// TIA Portal V20 export
DATA_BLOCK "InstStackMainDB"   // DB454
// stored: InstanceOfName 2200_StackMain, InstanceOfType FB
"2200_StackMain"
   // VAR_INPUT
   //    Calculate : Bool;
   //    SemiStep : Bool;
   //    FullStep : Bool;
   //    Auto : Bool;
   //    CycleStop : Bool;
   //    FastStop : Bool;
   //    Reset : Bool;
   //    Parameter : Struct
   //       Global : Struct
   //          CPM : LReal;
   //          StageWidth : LReal;
   //       END_STRUCT;
   //       "Step" : Struct
   //          MandrelUse : Bool;
   //          InitialPosFinalRoller : LReal;
   //          InitialPosCompensator : LReal;
   //       END_STRUCT;
   //       Auto : Struct
   //          SepaClean : Bool;
   //          CellCount : DInt;
   //          Compensator : Struct
   //             InitialPosCompensator : LReal;
   //          END_STRUCT;
   //          Anode : Struct
   //             PnPX1 : Struct
   //                InitialPosAnodePnPX1 : LReal;
   //                AnodePnPX1FwdOutputCam : Struct
   //                   OnPos : LReal;
   //                   OffPos : LReal;
   //                END_STRUCT;
   //                AnodePnPX1BwdOutputCam : Struct
   //                   OnPos : LReal;
   //                   OffPos : LReal;
   //                END_STRUCT;
   //                AnodeReelCutDataDeleteOffOutputCam : Struct
   //                   OnPos : LReal;
   //                   OffPos : LReal;
   //                END_STRUCT;
   //             END_STRUCT;
   //             PnPX2 : Struct
   //                InitialPosAnodePnPX2 : LReal;
   //                AnodePnPX2FwdOutputCam : Struct
   //                   OnPos : LReal;
   //                   OffPos : LReal;
   //                END_STRUCT;
   //                AnodePnPX2BwdOutputCam : Struct
   //                   OnPos : LReal;
   //                   OffPos : LReal;
   //                END_STRUCT;
   //             END_STRUCT;
   //             PnPZ1 : Struct
   //                InitialPosAnodePnPZ1 : LReal;
   //                AnodePnPZ1Down1OutputCam : Struct
   //                   OnPos : LReal;
   //                   OffPos : LReal;
   //                END_STRUCT;
   //                AnodePnPZ1Up1OutputCam : Struct
   //                   OnPos : LReal;
   //                   OffPos : LReal;
   //                END_STRUCT;
   //                AnodePnPZ1Down2OutputCam : Struct
   //                   OnPos : LReal;
   //                   OffPos : LReal;
   //                END_STRUCT;
   //                AnodePnPZ1Up2OutputCam : Struct
   //                   OnPos : LReal;
   //                   OffPos : LReal;
   //                END_STRUCT;
   //                AnodePnPZ1SuctionOnOutputCam : Struct
   //                   OnPos : LReal;
   //                   OffPos : LReal;
   //                END_STRUCT;
   //                AnodePnPZ1SuctionOffOutputCam : Struct
   //                   OnPos : LReal;
   //                   OffPos : LReal;
   //                END_STRUCT;
   //                AnodePnPZ1ReelCutBlowOutputCam : Struct
   //                   OnPos : LReal;
   //                   OffPos : LReal;
   //                END_STRUCT;
   //                AnodeAlignSuctionOnOutputCam : Struct
   //                   OnPos : LReal;
   //                   OffPos : LReal;
   //                END_STRUCT;
   //                AnodeReelCutDataDeleteOnOutputCam : Struct
   //                   OnPos : LReal;
   //                   OffPos : LReal;
   //                END_STRUCT;
   //                AnodeAlignVisionOutputCam : Struct
   //                   OnPos : LReal;
   //                   OffPos : LReal;
   //                END_STRUCT;
   //             END_STRUCT;
   //             PnPZ2 : Struct
   //                InitialPosAnodePnPZ2 : LReal;
   //                AnodePnPZ2Down1OutputCam : Struct
   //                   OnPos : LReal;
   //                   OffPos : LReal;
   //                END_STRUCT;
   //                AnodePnPZ2Up1OutputCam : Struct
   //                   OnPos : LReal;
   //                   OffPos : LReal;
   //                END_STRUCT;
   //                AnodePnPZ2Down2OutputCam : Struct
   //                   OnPos : LReal;
   //                   OffPos : LReal;
   //                END_STRUCT;
   //                AnodePnPZ2Up2OutputCam : Struct
   //                   OnPos : LReal;
   //                   OffPos : LReal;
   //                END_STRUCT;
   //                AnodePnPZ2SuctionOnOutputCam : Struct
   //                   OnPos : LReal;
   //                   OffPos : LReal;
   //                END_STRUCT;
   //                AnodePnPZ2SuctionOffOutputCam : Struct
   //                   OnPos : LReal;
   //                   OffPos : LReal;
   //                END_STRUCT;
   //                AnodeAlignSuctionOffOutputCam : Struct
   //                   OnPos : LReal;
   //                   OffPos : LReal;
   //                END_STRUCT;
   //             END_STRUCT;
   //          END_STRUCT;
   //          Cathode : Struct
   //             PnPX1 : Struct
   //                InitialPosCathodePnPX1 : LReal;
   //                CathodePnPX1FwdOutputCam : Struct
   //                   OnPos : LReal;
   //                   OffPos : LReal;
   //                END_STRUCT;
   //                CathodePnPX1BwdOutputCam : Struct
   //                   OnPos : LReal;
   //                   OffPos : LReal;
   //                END_STRUCT;
   //                CathodeReelCutDataDeleteOffOutputCam : Struct
   //                   OnPos : LReal;
   //                   OffPos : LReal;
   //                END_STRUCT;
   //             END_STRUCT;
   //             PnPX2 : Struct
   //                InitialPosCathodePnPX2 : LReal;
   //                CathodePnPX2FwdOutputCam : Struct
   //                   OnPos : LReal;
   //                   OffPos : LReal;
   //                END_STRUCT;
   //                CathodePnPX2BwdOutputCam : Struct
   //                   OnPos : LReal;
   //                   OffPos : LReal;
   //                END_STRUCT;
   //             END_STRUCT;
   //             PnPZ1 : Struct
   //                InitialPosCathodePnPZ1 : LReal;
   //                CathodePnPZ1Down1OutputCam : Struct
   //                   OnPos : LReal;
   //                   OffPos : LReal;
   //                END_STRUCT;
   //                CathodePnPZ1Up1OutputCam : Struct
   //                   OnPos : LReal;
   //                   OffPos : LReal;
   //                END_STRUCT;
   //                CathodePnPZ1Down2OutputCam : Struct
   //                   OnPos : LReal;
   //                   OffPos : LReal;
   //                END_STRUCT;
   //                CathodePnPZ1Up2OutputCam : Struct
   //                   OnPos : LReal;
   //                   OffPos : LReal;
   //                END_STRUCT;
   //                CathodePnPZ1SuctionOnOutputCam : Struct
   //                   OnPos : LReal;
   //                   OffPos : LReal;
   //                END_STRUCT;
   //                CathodePnPZ1SuctionOffOutputCam : Struct
   //                   OnPos : LReal;
   //                   OffPos : LReal;
   //                END_STRUCT;
   //                CathodePnPZ1ReelCutBlowOutputCam : Struct
   //                   OnPos : LReal;
   //                   OffPos : LReal;
   //                END_STRUCT;
   //                CathodeAlignSuctionOnOutputCam : Struct
   //                   OnPos : LReal;
   //                   OffPos : LReal;
   //                END_STRUCT;
   //                CathodeReelCutDataDeleteOnOutputCam : Struct
   //                   OnPos : LReal;
   //                   OffPos : LReal;
   //                END_STRUCT;
   //                CathodeAlignVisionOutputCam : Struct
   //                   OnPos : LReal;
   //                   OffPos : LReal;
   //                END_STRUCT;
   //             END_STRUCT;
   //             PnPZ2 : Struct
   //                InitialPosCathodePnPZ2 : LReal;
   //                CathodePnPZ2Down1OutputCam : Struct
   //                   OnPos : LReal;
   //                   OffPos : LReal;
   //                END_STRUCT;
   //                CathodePnPZ2Up1OutputCam : Struct
   //                   OnPos : LReal;
   //                   OffPos : LReal;
   //                END_STRUCT;
   //                CathodePnPZ2Down2OutputCam : Struct
   //                   OnPos : LReal;
   //                   OffPos : LReal;
   //                END_STRUCT;
   //                CathodePnPZ2Up2OutputCam : Struct
   //                   OnPos : LReal;
   //                   OffPos : LReal;
   //                END_STRUCT;
   //                CathodePnPZ2SuctionOnOutputCam : Struct
   //                   OnPos : LReal;
   //                   OffPos : LReal;
   //                END_STRUCT;
   //                CathodePnPZ2SuctionOffOutputCam : Struct
   //                   OnPos : LReal;
   //                   OffPos : LReal;
   //                END_STRUCT;
   //                CathodeAlignSuctionOffOutputCam : Struct
   //                   OnPos : LReal;
   //                   OffPos : LReal;
   //                END_STRUCT;
   //             END_STRUCT;
   //          END_STRUCT;
   //          FinalRoller : Struct
   //             InitialPosFinalRoller : LReal;
   //             FinalRollerFwdOutputCam : Struct
   //                OnPos : LReal;
   //                OffPos : LReal;
   //             END_STRUCT;
   //             FinalRollerBwdOutputCam : Struct
   //                OnPos : LReal;
   //                OffPos : LReal;
   //             END_STRUCT;
   //             FinalRollerStackTableDownOutputCam : Struct
   //                OnPos : LReal;
   //                OffPos : LReal;
   //             END_STRUCT;
   //             FinalRollerStackAnodeVisionOutputCam : Struct
   //                OnPos : LReal;
   //                OffPos : LReal;
   //             END_STRUCT;
   //             FinalRollerStackCathodeVisionOutputCam : Struct
   //                OnPos : LReal;
   //                OffPos : LReal;
   //             END_STRUCT;
   //          END_STRUCT;
   //          Mandrel : Struct
   //             InitialPosAnodeMandrelYFront : LReal;
   //             InitialPosAnodeMandrelYRear : LReal;
   //             InitialPosAnodeMandrelZFront : LReal;
   //             InitialPosAnodeMandrelZRear : LReal;
   //             InitialPosCathodeMandrelYFront : LReal;
   //             InitialPosCathodeMandrelYRear : LReal;
   //             InitialPosCathodeMandrelZFront : LReal;
   //             InitialPosCathodeMandrelZRear : LReal;
   //          END_STRUCT;
   //       END_STRUCT;
   //       StackCalculate : Struct
   //          Direction : Bool;
   //          RatioOption : Bool;
   //          TimeOption : Bool;
   //          PosOption : Bool;
   //          DoubleOption : Bool;
   //          StageHeight : LReal;
   //          StageGap : LReal;
   //          AccRatio : DInt;
   //          Ratio : Struct
   //             FinalRollerStart : LReal;
   //             FinalRollerEnd : LReal;
   //             PnPXStart : LReal;
   //             PnPXEnd : LReal;
   //             PnPZDownStart : LReal;
   //             PnPZDownEnd : LReal;
   //             PnPZUpStart : LReal;
   //             PnPZUpEnd : LReal;
   //             MandrelBwdStart : LReal;
   //             MandrelBwdEnd : LReal;
   //             MandrelFwdStart : LReal;
   //             MandrelFwdEnd : LReal;
   //             MandrelUpStart1 : LReal;
   //             MandrelUpEnd1 : LReal;
   //             MandrelUpStart2 : LReal;
   //             MandrelUpEnd2 : LReal;
   //             MandrelDownStart : LReal;
   //             MandrelDownEnd : LReal;
   //             MandrelYTerm : LReal;
   //             MandrelZTerm : LReal;
   //             MandrelBwdOffset : LReal;
   //             MandrelFwdOffset : LReal;
   //          END_STRUCT;
   //          "Time" : Struct
   //             FinalRollerStart : LReal;
   //             FinalRollerEnd : LReal;
   //             PnPXStart : LReal;
   //             PnPXEnd : LReal;
   //             PnPZDownStart : LReal;
   //             PnPZDownEnd : LReal;
   //             PnPZUpStart : LReal;
   //             PnPZUpEnd : LReal;
   //             MandrelBwdStart : LReal;
   //             MandrelBwdEnd : LReal;
   //             MandrelFwdStart : LReal;
   //             MandrelFwdEnd : LReal;
   //             MandrelUpStart1 : LReal;
   //             MandrelUpEnd1 : LReal;
   //             MandrelUpStart2 : LReal;
   //             MandrelUpEnd2 : LReal;
   //             MandrelDownStart : LReal;
   //             MandrelDownEnd : LReal;
   //          END_STRUCT;
   //          Position : Struct
   //             FinalRollerBwdPos : LReal;
   //             FinalRollerFwdPos : LReal;
   //          END_STRUCT;
   //          Distance : Struct
   //             Compensator : Struct
   //                Null : Bool;
   //             END_STRUCT;
   //             Anode : Struct
   //                PnPX1Distance : LReal;
   //                PnPX2Distance : LReal;
   //                PnPZ1Distance1 : LReal;
   //                PnPZ1Distance2 : LReal;
   //                PnPZ2Distance1 : LReal;
   //                PnPZ2Distance2 : LReal;
   //             END_STRUCT;
   //             Cathode : Struct
   //                PnPX1Distance : LReal;
   //                PnPX2Distance : LReal;
   //                PnPZ1Distance1 : LReal;
   //                PnPZ1Distance2 : LReal;
   //                PnPZ2Distance1 : LReal;
   //                PnPZ2Distance2 : LReal;
   //             END_STRUCT;
   //             FinalRoller : Struct
   //                Distance : LReal;
   //             END_STRUCT;
   //             Mandrel : Struct
   //                AnodeMandrelYFrontDistance : LReal;
   //                AnodeMandrelYRearDistance : LReal;
   //                CathodeMandrelYFrontDistance : LReal;
   //                CathodeMandrelYRearDistance : LReal;
   //                AnodeMandrelZFrontDistance : LReal;
   //                AnodeMandrelZRearDistance : LReal;
   //                CathodeMandrelZFrontDistance : LReal;
   //                CathodeMandrelZRearDistance : LReal;
   //             END_STRUCT;
   //          END_STRUCT;
   //       END_STRUCT;
   //    END_STRUCT;
   // END_VAR
   // VAR_OUTPUT
   //    Busy : Struct
   //       TotalBusy : Bool;
   //       CalculateBusy : Bool;
   //       SemiStepBusy : Bool;
   //       FullStepBusy : Bool;
   //       AutoBusy : Bool;
   //       CycleStopBusy : Bool;
   //       FastStopBusy : Bool;
   //       ResetBusy : Bool;
   //    END_STRUCT;
   //    Done : Struct
   //       TotalDone : Bool;
   //       CalculateDone : Bool;
   //       SemiStepDone : Bool;
   //       FullStepDone : Bool;
   //       AutoDone : Bool;
   //       CycleStopDone : Bool;
   //       FastStopDone : Bool;
   //       ResetDone : Bool;
   //    END_STRUCT;
   //    Error : Bool;
   //    ErrorID : DWord;
   //    SubNowStep : DInt;
   //    SubBeforeStep : DInt;
   //    OutputBits : Struct
   //       AnodePnP1Suction : Bool;
   //       AnodePnP1Blow : Bool;
   //       AnodePnP1ReelCutBlow : Bool;
   //       AnodePnP1RotaryWork : Bool;
   //       AnodePnP1RotaryHome : Bool;
   //       AnodeReelCutDataDelete : Bool;
   //       AnodePnP2Suction : Bool;
   //       AnodePnP2Blow : Bool;
   //       AnodeAlignSuction : Bool;
   //       AnodeAlignBlow : Bool;
   //       AnodeAlignVision : Bool;
   //       CathodePnP1Suction : Bool;
   //       CathodePnP1Blow : Bool;
   //       CathodePnP1ReelCutBlow : Bool;
   //       CathodePnP1RotaryWork : Bool;
   //       CathodePnP1RotaryHome : Bool;
   //       CathodeReelCutDataDelete : Bool;
   //       CathodePnP2Suction : Bool;
   //       CathodePnP2Blow : Bool;
   //       CathodeAlignSuction : Bool;
   //       CathodeAlignBlow : Bool;
   //       CathodeAlignVision : Bool;
   //       StackTableZAnodeDown : Bool;
   //       StackTableZCathodeDown : Bool;
   //       StackAnodeVision : Bool;
   //       StackCathodeVision : Bool;
   //    END_STRUCT;
   //    OutputData : Struct
   //       StackCellCount : DInt;
   //    END_STRUCT;
   // END_VAR
   // VAR_IN_OUT
   //    Axis : Struct
   //       MasterVirtual : DB_ANY;
   //       UnwinderVirtual : DB_ANY;
   //       UnwinderTop : DB_ANY;
   //       UnwinderBottom : DB_ANY;
   //       FinalRoller : DB_ANY;
   //       Compensator : DB_ANY;
   //       AnodePnPX1 : DB_ANY;
   //       AnodePnPX2 : DB_ANY;
   //       AnodePnPZ1 : DB_ANY;
   //       AnodePnPZ2 : DB_ANY;
   //       CathodePnPX1 : DB_ANY;
   //       CathodePnPX2 : DB_ANY;
   //       CathodePnPZ1 : DB_ANY;
   //       CathodePnPZ2 : DB_ANY;
   //       AnodeMandrelYFront : DB_ANY;
   //       AnodeMandrelYRear : DB_ANY;
   //       AnodeMandrelZFront : DB_ANY;
   //       AnodeMandrelZRear : DB_ANY;
   //       CathodeMandrelYFront : DB_ANY;
   //       CathodeMandrelYRear : DB_ANY;
   //       CathodeMandrelZFront : DB_ANY;
   //       CathodeMandrelZRear : DB_ANY;
   //       SepaGripperX : DB_ANY;
   //    END_STRUCT;
   //    Cam : Struct
   //       FinalRollerCam : DB_ANY;
   //       CompensatorCam : DB_ANY;
   //       AnodePnPX1Cam : DB_ANY;
   //       AnodePnPX2Cam : DB_ANY;
   //       AnodePnPZ1Cam : DB_ANY;
   //       AnodePnPZ2Cam : DB_ANY;
   //       CathodePnPX1Cam : DB_ANY;
   //       CathodePnPX2Cam : DB_ANY;
   //       CathodePnPZ1Cam : DB_ANY;
   //       CathodePnPZ2Cam : DB_ANY;
   //       AnodeMandrelYFrontCam : DB_ANY;
   //       AnodeMandrelYRearCam : DB_ANY;
   //       AnodeMandrelZFrontCam : DB_ANY;
   //       AnodeMandrelZRearCam : DB_ANY;
   //       CathodeMandrelYFrontCam : DB_ANY;
   //       CathodeMandrelYRearCam : DB_ANY;
   //       CathodeMandrelZFrontCam : DB_ANY;
   //       CathodeMandrelZRearCam : DB_ANY;
   //    END_STRUCT;
   //    OutputCam : Struct
   //       FinalRollerXFwdOutputCam : DB_ANY;
   //       FinalRollerXBwdOutputCam : DB_ANY;
   //       FinalRollerXStackTableDownOutputCam : DB_ANY;
   //       FinalRollerXStackAnodeVisionOutputCam : DB_ANY;
   //       FinalRollerXStackCathodeVisionOutputCam : DB_ANY;
   //       AnodePnPX1FwdOutputCam : DB_ANY;
   //       AnodePnPX1BwdOutputCam : DB_ANY;
   //       AnodePnPX2FwdOutputCam : DB_ANY;
   //       AnodePnPX2BwdOutputCam : DB_ANY;
   //       AnodePnPZ1Down1OutputCam : DB_ANY;
   //       AnodePnPZ1Up1OutputCam : DB_ANY;
   //       AnodePnPZ2Down1OutputCam : DB_ANY;
   //       AnodePnPZ2Up1OutputCam : DB_ANY;
   //       AnodePnPZ1Down2OutputCam : DB_ANY;
   //       AnodePnPZ1Up2OutputCam : DB_ANY;
   //       AnodePnPZ2Down2OutputCam : DB_ANY;
   //       AnodePnPZ2Up2OutputCam : DB_ANY;
   //       AnodePnPZ1SuctionOnOutputCam : DB_ANY;
   //       AnodePnPZ1SuctionOffOutputCam : DB_ANY;
   //       AnodePnPZ1ReelCutBlowOutputCam : DB_ANY;
   //       AnodePnPZ2SuctionOnOutputCam : DB_ANY;
   //       AnodePnPZ2SuctionOffOutputCam : DB_ANY;
   //       AnodeAlignSuctionOnOutputCam : DB_ANY;
   //       AnodeAlignSuctionOffOutputCam : DB_ANY;
   //       AnodePnPZ1ReelCutDataDeleteOnOutputCam : DB_ANY;
   //       AnodePnP1XReelCutDataDeleteOffOutputCam : DB_ANY;
   //       AnodeAlignVisionOutputCam : DB_ANY;
   //       CathodePnPX1FwdOutputCam : DB_ANY;
   //       CathodePnPX1BwdOutputCam : DB_ANY;
   //       CathodePnPX2FwdOutputCam : DB_ANY;
   //       CathodePnPX2BwdOutputCam : DB_ANY;
   //       CathodePnPZ1Down1OutputCam : DB_ANY;
   //       CathodePnPZ1Up1OutputCam : DB_ANY;
   //       CathodePnPZ2Down1OutputCam : DB_ANY;
   //       CathodePnPZ2Up1OutputCam : DB_ANY;
   //       CathodePnPZ1Down2OutputCam : DB_ANY;
   //       CathodePnPZ1Up2OutputCam : DB_ANY;
   //       CathodePnPZ2Down2OutputCam : DB_ANY;
   //       CathodePnPZ2Up2OutputCam : DB_ANY;
   //       CathodePnPZ1SuctionOnOutputCam : DB_ANY;
   //       CathodePnPZ1SuctionOffOutputCam : DB_ANY;
   //       CathodePnPZ1ReelCutBlowOutputCam : DB_ANY;
   //       CathodePnPZ2SuctionOnOutputCam : DB_ANY;
   //       CathodePnPZ2SuctionOffOutputCam : DB_ANY;
   //       CathodeAlignSuctionOnOutputCam : DB_ANY;
   //       CathodeAlignSuctionOffOutputCam : DB_ANY;
   //       CathodePnPZ1ReelCutDataDeleteOnOutputCam : DB_ANY;
   //       CathodePnP1XReelCutDataDeleteOffOutputCam : DB_ANY;
   //       CathodeAlignVisionOutputCam : DB_ANY;
   //    END_STRUCT;
   //    ReelcutInterface : Struct
   //       AutoStandBy : Bool;
   //       AnodeReelcutStandby : Bool;
   //       AnodeReelcutStart : Bool;
   //       AnodeReelcutDone : Bool;
   //       CathodeReelcutStandby : Bool;
   //       CathodeReelcutStart : Bool;
   //       CathodeReelcutDone : Bool;
   //    END_STRUCT;
   //    CalculateInterface : Struct
   //       Execute : Bool;
   //       Done : Bool;
   //       Busy : Bool;
   //       Error : Bool;
   //       ErrorID : DWord;
   //       NowCmd : DInt;
   //       BeforeCmd : DInt;
   //    END_STRUCT;
   // END_VAR
   // VAR
   //    statNowCmd : DInt;
   //    statBeforeCmd : DInt;
   //    statDone : Bool;
   //    statTimeTable : Array[1..50] of Time;
   //    statStartTime : Time;
   //    statEndTime : Time;
   //    instTriggerCalculate : R_TRIG;
   //    instTriggerSemiStep { S7_SetPoint := 'True'} : R_TRIG;
   //    instTriggerFullStep { S7_SetPoint := 'True'} : R_TRIG;
   //    instTriggerAuto { S7_SetPoint := 'True'} : R_TRIG;
   //    instTriggerStop { S7_SetPoint := 'True'} : R_TRIG;
   //    instTriggerReset { S7_SetPoint := 'True'} : R_TRIG;
   //    instStackSemiStep { S7_SetPoint := 'True'} : "2202_StackSemiStep";
   //    instStackFullStepAuto { S7_SetPoint := 'True'} : "2203_StackFullStepAuto";
   //    instStackStop { S7_SetPoint := 'True'} : "2204_StackStop";
   //    instStackReset { S7_SetPoint := 'True'} : "2205_StackReset";
   //    instOutputControl { S7_SetPoint := 'True'} : "2206_OutputControl";
   // END_VAR
BEGIN
END_DATA_BLOCK
